// TIA Portal V18 export
DATA_BLOCK "数据块_1"   // DB2
{ S7_Optimized_Access := 'TRUE' }
VERSION : 0.1
// stored: AutoNumber true, DBAccessibleFromOPCUA true, IsOnlyStoredInLoadMemory false, IsRetainMemResEnabled false, IsWriteProtectedInAS false, MemoryReserve 100
   VAR
      Room1_Interlock : Bool;
      Room2_Interlock : Bool;
      ACC_Interlock : Bool;
      VerticalBeam_Interlock : Bool;
      Interlock : Bool;
   END_VAR
BEGIN
END_DATA_BLOCK
